(* IEC 61131-3 sources: Industry-PLC-LLM/data/PLCBEAD_repo/PLCBEAD_PLCEmbed-main/PLC-BEAD/Source/GEB/F_LIN2, 1 file *)

(* ---- F_LIN2.ST ---- *)
FUNCTION F_LIN2:REAL
	VAR_INPUT
		X :	REAL;
		X1 :	REAL;
		Y1 :	REAL;
		X2 :	REAL;
		Y2 :	REAL;
	END_VAR

	F_LIN2 := (Y2 - Y1) / (X2 - X1) * (X - X1) + Y1;

END_FUNCTION

PROGRAM program0
  VAR
    LocalVar0 : REAL;
	LocalVaR1  : REAL;
	LocalVaR2 : REAL;
	LocalVar3 : REAL;
	LocalVar4 : REAL;
	  LocalOUT  : REAL;
  END_VAR
  	LocalOUT := F_LIN2(LocalVar0, LocalVaR1 , LocalVaR2, LocalVar3, LocalVar4);
END_PROGRAM
